FUNCTION_BLOCK Test_TStreamAdd_Read_LINT EXTENDS T_UnitTestBase
VAR
    Stream  : T_Stream(StreamLength := 2);
    ArgType : E_ArgTypeId := E_ArgTypeId.Type_LINT;
END_VAR

Stream.Init(2);

// add a LINT...
Stream.SetNextArgTypeId(ArgType);
Stream.Add_LINT(123456789);

Stream.SetReadPosition(0);

// check next arg type is correct...
Assertion.AssertEquals_INT(Expected     := ArgType,
                           Actual       := Stream.GetNextArgTypeId(),
                           VariableName := 'Stream.GetNextArgTypeId()');

// check next value...	
Assertion.AssertEquals_LINT(Expected     := 123456789,
                            Actual       := Stream.Read_LINT(),
                            VariableName := 'Stream.Read_LINT()');

// check we are at the end of the stream..							
Assertion.AssertEquals_UDINT(Expected     := Stream.StreamLength,
                             Actual       := Stream.ReadPosition,
                             VariableName := 'Stream.ReadPosition');

TestFinished();

END_FUNCTION_BLOCK

(* stored: Version 1.1.0.1, ProductVersion 3.1.4024.9
   POU Test_TStreamAdd_Read_LINT: Id {d2743c81-1757-4e56-b58a-a365855abc4d}, SpecialFunc None *)
